% RSLogix 500 project PRACTICE JSR 1.20.11.RSS, saved by version 8.30.00.15 %
PROJECT "UNTITLED"    % processor: MicroLogix 1000 %

PROGRAM FILES
  LAD 2 "MAIN_PROG"  3 rungs
  LAD 3 "USER_FAULT"  7 rungs
  LAD 4 "HSC_INT"  7 rungs
  LAD 5 "STI_INT"  1 rungs
  LAD 6, 7, 8, 9, 10, 11, 12, 13, 14, 15, 16: only END

DATA FILES
  O0 OUTPUT  1 elements
  I1 INPUT  2 elements
  S2 STATUS  33 elements
  B3 BINARY  32 elements
  T4 TIMER  40 elements
  C5 COUNTER  32 elements
  R6 CONTROL  16 elements
  N7 INTEGER  105 elements

LADDER 2 "MAIN_PROG"
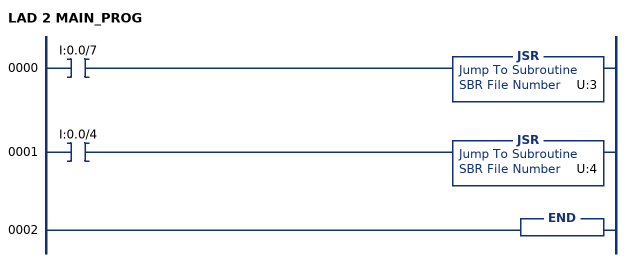
% Rung: 0 %
SOR XIC I:0.0/7 JSR U:3 EOR
% Rung: 1 %
SOR XIC I:0.0/4 JSR U:4 EOR
% Rung: 2 %
SOR END EOR

LADDER 3 "USER_FAULT"
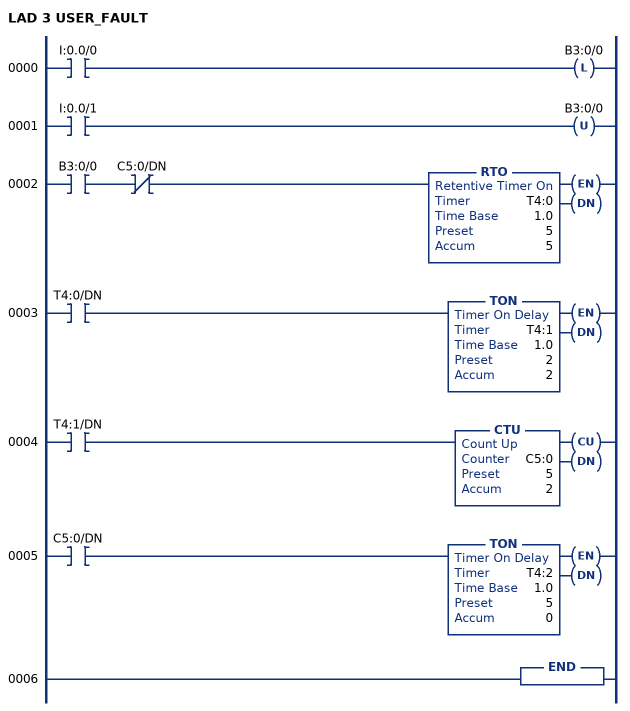
% Rung: 0 %
SOR XIC I:0.0/0 OTL B3:0/0 EOR
% Rung: 1 %
SOR XIC I:0.0/1 OTU B3:0/0 EOR
% Rung: 2 %
SOR XIC B3:0/0 XIO C5:0/DN RTO T4:0 1.0 5 5 EOR
% Rung: 3 %
SOR XIC T4:0/DN TON T4:1 1.0 2 2 EOR
% Rung: 4 %
SOR XIC T4:1/DN CTU C5:0 5 2 EOR
% Rung: 5 %
SOR XIC C5:0/DN TON T4:2 1.0 5 0 EOR
% Rung: 6 %
SOR END EOR

LADDER 4 "HSC_INT"
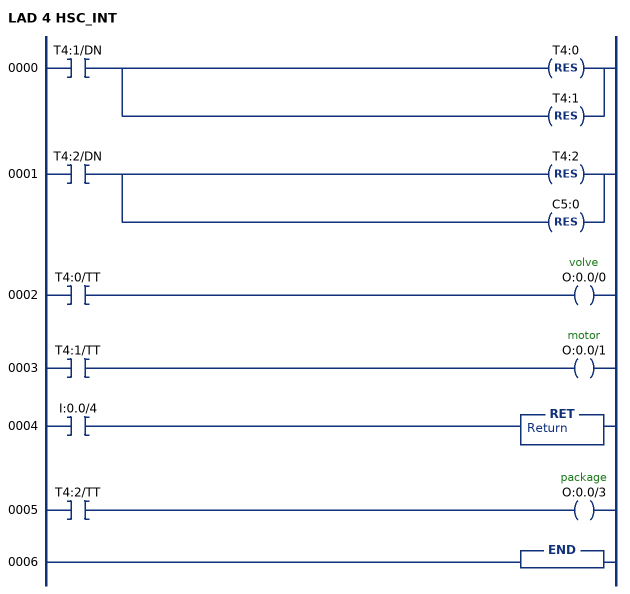
% Rung: 0 %
SOR XIC T4:1/DN BST RES T4:0 NXB RES T4:1 BND EOR
% Rung: 1 %
SOR XIC T4:2/DN BST RES T4:2 NXB RES C5:0 BND EOR
% Rung: 2 %
SOR XIC T4:0/TT OTE O:0.0/0 EOR
%   O:0.0/0  "volve" %
% Rung: 3 %
SOR XIC T4:1/TT OTE O:0.0/1 EOR
%   O:0.0/1  "motor" %
% Rung: 4 %  % edit flag set %
SOR XIC I:0.0/4 RET EOR
% Rung: 5 %
SOR XIC T4:2/TT OTE O:0.0/3 EOR
%   O:0.0/3  "package" %
% Rung: 6 %
SOR END EOR

DATA TABLE (non-zero values as saved)
DATA B3
% B3:0 % 0X0001 0X0000 0X0000 0X0000 0X0000 0X0000 0X0000 0X0000 0X0000 0X0000
DATA T4
% .PRE .ACC %
% T4:0 % 5 5
% T4:1 % 2 2
% T4:2 % 5 0
DATA C5
% .PRE .ACC %
% C5:0 % 5 2
